// TIA Portal project "EJERCICIO 23" (V11)

(* hardware
DEVICE "S7300/ET200 station_1"  SIMATIC 300-Station
   slot 0: "Perfil soporte_0"  Rail  6ES7 390-1***0-0AA0
   slot 2: "PLC_1"  CPU 313C-2 DP  6ES7 313-6CF03-0AB0  V2.6
      slot 0: "Interfaz MPI_1"  MPI
      slot 1: "Interfaz DP_1"  DP
      slot 2: "DI16/DO16_1"  DI16/DO16
      slot 4: "Contaje_1"  Counter
*)

// ===== PLC "PLC_1"  CPU 313C-2 DP =====

VAR_GLOBAL   // PLC tag table "Tabla de variables estándar"
   "CAFE SOLO" AT %I0.0 : Bool;
   "CAFE EXPRESSO" AT %I0.1 : Bool;
   "CAFE CON LECHE" AT %I0.2 : Bool;
   "LECHE" AT %I0.3 : Bool;
   "TE" AT %I0.4 : Bool;
   "AGUA" AT %I0.5 : Bool;
   "V CAFE" AT %Q0.0 : Bool;
   "V LECHE" AT %Q0.1 : Bool;
   "V TE" AT %Q0.2 : Bool;
   "V AGUA" AT %Q0.3 : Bool;
   "MONEDAS" AT %I0.6 : Bool;
   "Tag_1" AT %MB0 : Byte;
   "Tag_2" AT %M0.0 : Bool;
   "Tag_3" AT %T0 : Timer;
   "Tag_4" AT %M0.1 : Bool;
   "Tag_5" AT %M0.2 : Bool;
   "Tag_6" AT %M0.3 : Bool;
   "Tag_7" AT %M0.4 : Bool;
   "Tag_8" AT %M0.5 : Bool;
   "Tag_9" AT %T1 : Timer;
   "Tag_10" AT %M0.6 : Bool;
   "Tag_11" AT %T2 : Timer;
   "Tag_12" AT %M0.7 : Bool;
   "Tag_13" AT %T3 : Timer;
   "Tag_14" AT %T4 : Timer;
   "Tag_15" AT %T5 : Timer;
   "Tag_16" AT %T6 : Timer;
END_VAR

DATA_BLOCK "AUXILIARES"   // DB1
{ S7_Optimized_Access := 'FALSE' }
VERSION : 0.1
   VAR
      FLANCOS : Array [0..14] of Bool;
      BOBINAS : Array [0..7] of Bool;
      CONTADOR : Array [0..0] of Int;
   END_VAR
BEGIN
END_DATA_BLOCK

ORGANIZATION_BLOCK "Main"   // OB1, LAD
TITLE = "Main Program Sweep (Cycle)"
{ S7_Optimized_Access := 'FALSE' }
VERSION : 0.1
// MAQUINA ESPENDEDORA DE CAFE.
   VAR_TEMP
      OB1_EV_CLASS : Byte;   // Bits 0-3 = 1 (Coming event), Bits 4-7 = 1 (Event class 1)
      OB1_SCAN_1 : Byte;   // 1 (Cold restart scan 1 of OB 1), 3 (Scan 2-n of OB 1)
      OB1_PRIORITY : Byte;   // Priority of OB Execution
      OB1_OB_NUMBR : Byte;   // 1 (Organization block 1, OB1)
      OB1_RESERVED_1 : Byte;   // Reserved for system
      OB1_RESERVED_2 : Byte;   // Reserved for system
      OB1_PREV_CYCLE : Int;   // Cycle time of previous OB1 scan (milliseconds)
      OB1_MIN_CYCLE : Int;   // Minimum cycle time of OB1 (milliseconds)
      OB1_MAX_CYCLE : Int;   // Maximum cycle time of OB1 (milliseconds)
      OB1_DATE_TIME : Date_And_Time;   // Date and time OB1 started
   END_VAR
BEGIN
END_ORGANIZATION_BLOCK